// TwinCAT 3 PLC project FastLog
// ProgramVersion: 3.1.4024.0
// libraries:
//   Tc2_Standard, * (Beckhoff Automation GmbH)
//   Tc2_System, * (Beckhoff Automation GmbH)
//   Tc2_Utilities, * (Beckhoff Automation GmbH)
//   Tc3_Module, * (Beckhoff Automation GmbH)
// project tree:
//   / FileLogger.TcTTO, FastSample.TcTTO
//   GVLs/ GVL.TcGVL, SENSOR_LIST.TcGVL
//   POUs/ F_TimeStructToUnixMs.TcPOU, PRG_FileLogger.TcPOU, PRG_FastSample.TcPOU
// real-time tasks:
//   TASK FastSample: cycle T#100us, priority 20, ADS port 350
//   TASK FileLogger: cycle T#1ms, priority 10, ADS port 351
// I/O:
//   DEVICE Device 1 (Beckhoff CCAT)
//   DEVICE Device 2 (EtherCAT), AmsNetId 5.156.10.9.3.1
//     Term 1 (EK1200) [EK1200-5000 EtherCAT Power supply (2A E-Bus)]
//       Term 2 (EL1809) [EL1809 16Ch. Dig. Input 24V, 3ms]
//       Term 3 (EL1889) [EL1889 16Ch. Dig. Input 24V, 3ms, negative]
//       Term 4 (EL2008) [EL2008 8Ch. Dig. Output 24V, 0.5A]
//       Term 5 (EL2008) [EL2008 8Ch. Dig. Output 24V, 0.5A]
//       Term 6 (EL2008) [EL2008 8Ch. Dig. Output 24V, 0.5A]
//       Term 7 (EL2634) [EL2634 4Ch. Relay Output, NO (250V AC / 30V DC)]
//       Term 8 (EL2889) [EL2889 16Ch. Dig. Output 24V, 0.5A, negative]
//       Term 9 (EL2809) [EL2809 16Ch. Dig. Output 24V, 0.5A]
//       Term 10 (EL9011) [EL9011 End Terminal]
//   DEVICE Device 5 (EtherCAT), AmsNetId 5.156.10.9.6.1
//     Term 11 (EK1100) [EK1100 EtherCAT Coupler (2A E-Bus)]
//       Term 12 (EL5151) [EL5151 1Ch. Inc. Encoder]
//       Term 13 (EL5151) [EL5151 1Ch. Inc. Encoder]
//       Term 14 (EL3182) [EL3182 2Ch. Ana. Input 4-20mA, HART]
//         modules: Ch. 1, Ch. 2, Ch. 1, Ch. 1, Ch. 1, Ch. 1, Ch. 1, Ch. 1, Ch. 1, Ch. 1, Ch. 1, Ch. 1, Ch. 1, Ch. 1, Ch. 1
//       Term 15 (EL3182) [EL3182 2Ch. Ana. Input 4-20mA, HART]
//         modules: Ch. 1, Ch. 2, Ch. 1, Ch. 1, Ch. 1, Ch. 1, Ch. 1, Ch. 1, Ch. 1, Ch. 1, Ch. 1, Ch. 1, Ch. 1, Ch. 1, Ch. 1
//       Term 6 (EL6731) [EL6731 PROFIBUS DP Master]
//       Term 7 (EL6751) [EL6751 CANopen Master]
//       Term 18 (EL6022) [EL6022 Interface 2Ch. (RS422/485)]
//       Term 19 (EL6022) [EL6022 Interface 2Ch. (RS422/485)]
//       Term 62 (EL9011) [EL9011 End Terminal]
//     Term 20 (EK1100) [EK1100 EtherCAT Coupler (2A E-Bus)]
//       Term 21 (EL3201-0020) [EL3201-0020 1Ch. Ana. Input PT100 (RTD), High Precision, calibrated]
//       Term 22 (EL3201-0020) [EL3201-0020 1Ch. Ana. Input PT100 (RTD), High Precision, calibrated]
//       Term 23 (EL3201-0020) [EL3201-0020 1Ch. Ana. Input PT100 (RTD), High Precision, calibrated]
//       Term 24 (EL3201-0020) [EL3201-0020 1Ch. Ana. Input PT100 (RTD), High Precision, calibrated]
//       Term 25 (EL3201-0020) [EL3201-0020 1Ch. Ana. Input PT100 (RTD), High Precision, calibrated]
//       Term 26 (EL3201-0020) [EL3201-0020 1Ch. Ana. Input PT100 (RTD), High Precision, calibrated]
//       Term 27 (EL3201-0020) [EL3201-0020 1Ch. Ana. Input PT100 (RTD), High Precision, calibrated]
//       Term 28 (EL3201-0020) [EL3201-0020 1Ch. Ana. Input PT100 (RTD), High Precision, calibrated]
//       Term 29 (EL3201-0020) [EL3201-0020 1Ch. Ana. Input PT100 (RTD), High Precision, calibrated]
//       Term 30 (EL9410) [EL9410 E-Bus Power Supplier  (Diagnostics)]
//       Term 31 (EL3201-0020) [EL3201-0020 1Ch. Ana. Input PT100 (RTD), High Precision, calibrated]
//       Term 32 (EL3201-0020) [EL3201-0020 1Ch. Ana. Input PT100 (RTD), High Precision, calibrated]
//       Term 33 (EL3201-0020) [EL3201-0020 1Ch. Ana. Input PT100 (RTD), High Precision, calibrated]
//       Term 34 (EL3201-0020) [EL3201-0020 1Ch. Ana. Input PT100 (RTD), High Precision, calibrated]
//       Term 35 (EL3201-0020) [EL3201-0020 1Ch. Ana. Input PT100 (RTD), High Precision, calibrated]
//       Term 36 (EL3201-0020) [EL3201-0020 1Ch. Ana. Input PT100 (RTD), High Precision, calibrated]
//       Term 37 (EL3201-0020) [EL3201-0020 1Ch. Ana. Input PT100 (RTD), High Precision, calibrated]
//       Term 38 (EL3218) [EL3218-0000 8Ch. Ana. Input PT100 (RTD)]
//       Term 39 (EL3218) [EL3218-0000 8Ch. Ana. Input PT100 (RTD)]
//       Term 40 (EL3218) [EL3218-0000 8Ch. Ana. Input PT100 (RTD)]
//       Term 41 (EL9410) [EL9410 E-Bus Power Supplier  (Diagnostics)]
//       Term 42 (EL3218) [EL3218-0000 8Ch. Ana. Input PT100 (RTD)]
//       Term 43 (EL3218) [EL3218-0000 8Ch. Ana. Input PT100 (RTD)]
//       Term 44 (EL3218) [EL3218-0000 8Ch. Ana. Input PT100 (RTD)]
//       Term 45 (EL3214) [EL3214 4Ch. Ana. Input PT100 (RTD)]
//       Term 46 (EL4124) [EL4124 4Ch. Ana. Output 4-20mA, 16bit]
//       Term 47 (EL4124) [EL4124 4Ch. Ana. Output 4-20mA, 16bit]
//       Term 48 (EL4124) [EL4124 4Ch. Ana. Output 4-20mA, 16bit]
//       Term 49 (EL4124) [EL4124 4Ch. Ana. Output 4-20mA, 16bit]
//       Term 50 (EL4124) [EL4124 4Ch. Ana. Output 4-20mA, 16bit]
//       Term 51 (EL4124) [EL4124 4Ch. Ana. Output 4-20mA, 16bit]
//       Term 52 (EL4124) [EL4124 4Ch. Ana. Output 4-20mA, 16bit]
//       Term 53 (EL3356) [EL3356 1Ch. Ana. Input Resistor Bridge Terminal, 16bit, High Precision]
//       Term 63 (EL9011) [EL9011 End Terminal]
//     Term 54 (EK1100) [EK1100 EtherCAT Coupler (2A E-Bus)]
//       Term 55 (ELM3148-0000) [ELM3148-0000 8Ch. Ana. Input +/-10V, +/-20mA, 24 bit, high precision]
//       Term 56 (ELM3148-0000) [ELM3148-0000 8Ch. Ana. Input +/-10V, +/-20mA, 24 bit, high precision]
//       Term 57 (ELM3148-0000) [ELM3148-0000 8Ch. Ana. Input +/-10V, +/-20mA, 24 bit, high precision]
//       Term 58 (ELM3148-0000) [ELM3148-0000 8Ch. Ana. Input +/-10V, +/-20mA, 24 bit, high precision]
//       Term 59 (ELM3148-0000) [ELM3148-0000 8Ch. Ana. Input +/-10V, +/-20mA, 24 bit, high precision]
//       Term 60 (ELM3148-0000) [ELM3148-0000 8Ch. Ana. Input +/-10V, +/-20mA, 24 bit, high precision]
//       Term 61 (EL9410) [EL9410 E-Bus Power Supplier  (Diagnostics)]
//       Term 62 (ELM3148-0000) [ELM3148-0000 8Ch. Ana. Input +/-10V, +/-20mA, 24 bit, high precision]
//       Term 63 (ELM3148-0000) [ELM3148-0000 8Ch. Ana. Input +/-10V, +/-20mA, 24 bit, high precision]
//       Term 64 (ELM3148-0000) [ELM3148-0000 8Ch. Ana. Input +/-10V, +/-20mA, 24 bit, high precision]
//       Term 65 (ELM3148-0000) [ELM3148-0000 8Ch. Ana. Input +/-10V, +/-20mA, 24 bit, high precision]
//       Term 66 (ELM3148-0000) [ELM3148-0000 8Ch. Ana. Input +/-10V, +/-20mA, 24 bit, high precision]
//       Term 67 (ELM3148-0000) [ELM3148-0000 8Ch. Ana. Input +/-10V, +/-20mA, 24 bit, high precision]
//       Term 68 (EL9410) [EL9410 E-Bus Power Supplier  (Diagnostics)]
//       Term 69 (ELM3148-0000) [ELM3148-0000 8Ch. Ana. Input +/-10V, +/-20mA, 24 bit, high precision]
//       Term 70 (ELM3148-0000) [ELM3148-0000 8Ch. Ana. Input +/-10V, +/-20mA, 24 bit, high precision]
//       Term 71 (ELM3148-0000) [ELM3148-0000 8Ch. Ana. Input +/-10V, +/-20mA, 24 bit, high precision]
//       Term 64 (EL9011) [EL9011 End Terminal]
//   DEVICE Device 6 (USB)
//     Box 1 (CX2100 Power Supply)
//   DEVICE Device 7 (NOV-DP-RAM)
//   DEVICE Device 3 (EL6731), AmsNetId 5.156.10.9.4.1
//   DEVICE Device 4 (EL6751), AmsNetId 5.156.10.9.5.1
// variable links:
//   FastLog/FastLog Instance <-> Device 5 (EtherCAT)/Term 54 (EK1100)/Term 55 (ELM3148-0000)
//     FastSample Inputs/SENSOR_LIST.AInput_{1..8} <-> PAI Samples 1 Channel {1..8}/Samples[0]  (8 links)
//   FastLog/FastLog Instance <-> Device 5 (EtherCAT)/Term 54 (EK1100)/Term 56 (ELM3148-0000)
//     FastSample Inputs/SENSOR_LIST.AInput_{9..16} <-> PAI Samples 1 Channel {1..8}/Samples[0]  (8 links)
//   FastLog/FastLog Instance <-> Device 5 (EtherCAT)/Term 54 (EK1100)/Term 57 (ELM3148-0000)
//     FastSample Inputs/SENSOR_LIST.AInput_17 <-> PAI Samples 1 Channel 1/Samples[0]
//     FastSample Inputs/SENSOR_LIST.AInput_18 <-> PAI Samples 1 Channel 2/Samples[0]
//     FastSample Inputs/SENSOR_LIST.AInput_19 <-> PAI Samples 1 Channel 3/Samples[0]
//     FastSample Inputs/SENSOR_LIST.AInput_20 <-> PAI Samples 1 Channel 4/Samples[0]
//     FastSample Inputs/SENSOR_LIST.AInput_21 <-> PAI Samples 1 Channel 5/Samples[0]
//     FastSample Inputs/SENSOR_LIST.AInput_22 <-> PAI Samples 1 Channel 6/Samples[0]
//     FastSample Inputs/SENSOR_LIST.AInput_24 <-> PAI Samples 1 Channel 8/Samples[0]
//     FastSample Inputs/SENSOR_LIST.AInput_23 <-> PAI Samples 1 Channel 7/Samples

CONFIGURATION FastLog
    RESOURCE PLC ON TwinCAT3
        TASK FileLogger(INTERVAL := T#100us, PRIORITY := 20);
        TASK FastSample(INTERVAL := T#1ms, PRIORITY := 10);
        PROGRAM PRG_FileLogger WITH FileLogger : PRG_FileLogger;
        PROGRAM PRG_FastSample WITH FastSample : PRG_FastSample;
    END_RESOURCE
END_CONFIGURATION

// ---- GVLs/GVL.TcGVL
VAR_GLOBAL CONSTANT
    C_BUFFER_SIZE : UDINT := 100000;   // buffer satır sayısı (ihtiyacına göre büyüt)
    C_NUM_SENSORS : UINT  := 60;       // sende 60 sensör var demiştin
END_VAR


VAR_GLOBAL
    // Start/Stop
    g_bLogStart       : BOOL := FALSE;
    g_bLogStop        : BOOL := FALSE;
    g_bLogging        : BOOL := FALSE;

    // Epoch ms (sampler doldurur)
    g_epochMs        : ULINT := 0;
	g_epochBaseMs    : ULINT := 0;   // log start anındaki gerçek epoch(ms)
    g_epochOffsetMs  : UDINT := 0; 

    // Ring buffer
    g_aTimeBuffer     : ARRAY[0..C_BUFFER_SIZE-1] OF ULINT;
    g_aValBuffer      : ARRAY[0..C_BUFFER_SIZE-1, 1..C_NUM_SENSORS] OF LREAL;

    g_wrIndex         : UDINT := 0;
    g_rdIndex         : UDINT := 0;
    g_bufferUsed      : UDINT := 0;
    g_bufferOverflow  : BOOL  := FALSE;

    // Sampler burayı dolduracak
    g_arCurrentValues : ARRAY[1..C_NUM_SENSORS] OF LREAL;

    // Dosya yolu / isim
    g_sBasePath       : STRING(255) := 'D:\';   // istediğin klasör
    g_sFileName       : STRING(64);
    g_sPath           : STRING(320);

    // Yazma kontrol
    g_headerPending   : BOOL := FALSE;
    g_lineReady       : BOOL := FALSE;

    // Chunk buffer (data satırları buraya toplanır)
    g_sLine           : STRING(16384);

END_VAR

// ---- GVLs/SENSOR_LIST.TcGVL
VAR_GLOBAL
	
	AInput_1  AT %I* : DINT;
	AInput_2  AT %I* : DINT;
	AInput_3  AT %I* : DINT;
	AInput_4  AT %I* : DINT;
	AInput_5  AT %I* : DINT;
	AInput_6  AT %I* : DINT;
	AInput_7  AT %I* : DINT;
	AInput_8  AT %I* : DINT;
	AInput_9  AT %I* : DINT;
	AInput_10 AT %I* : DINT;
	AInput_11 AT %I* : DINT;
	AInput_12 AT %I* : DINT;
	AInput_13 AT %I* : DINT;
	AInput_14 AT %I* : DINT;
	AInput_15 AT %I* : DINT;
	AInput_16 AT %I* : DINT;
	AInput_17 AT %I* : DINT;
	AInput_18 AT %I* : DINT;
	AInput_19 AT %I* : DINT;
	AInput_20 AT %I* : DINT;
	
	AInput_21 AT %I* : DINT;
	AInput_22 AT %I* : DINT;
	AInput_23 AT %I* : DINT;
	AInput_24 AT %I* : DINT;
	AInput_25 AT %I* : DINT;
	AInput_26 AT %I* : DINT;
	AInput_27 AT %I* : DINT;
	AInput_28 AT %I* : DINT;
	AInput_29 AT %I* : DINT;
	AInput_30 AT %I* : DINT;
	
	AInput_31 AT %I* : DINT;
	AInput_32 AT %I* : DINT;
	AInput_33 AT %I* : DINT;
	AInput_34 AT %I* : DINT;
	AInput_35 AT %I* : DINT;
	AInput_36 AT %I* : DINT;
	AInput_37 AT %I* : DINT;
	AInput_38 AT %I* : DINT;
	AInput_39 AT %I* : DINT;
	AInput_40 AT %I* : DINT;
	
	AInput_41 AT %I* : DINT;
	AInput_42 AT %I* : DINT;
	AInput_43 AT %I* : DINT;
	AInput_44 AT %I* : DINT;
	AInput_45 AT %I* : DINT;
	AInput_46 AT %I* : DINT;
	AInput_47 AT %I* : DINT;
	AInput_48 AT %I* : DINT;
	AInput_49 AT %I* : DINT;
	AInput_50 AT %I* : DINT;
	
	AInput_51 AT %I* : DINT;
	AInput_52 AT %I* : DINT;
	AInput_53 AT %I* : DINT;
	AInput_54 AT %I* : DINT;
	AInput_55 AT %I* : DINT;
	AInput_56 AT %I* : DINT;
	AInput_57 AT %I* : DINT;
	AInput_58 AT %I* : DINT;
	AInput_59 AT %I* : DINT;
	AInput_60 AT %I* : DINT;

END_VAR

// ---- POUs/PRG_FileLogger.TcPOU
PROGRAM PRG_FileLogger
VAR
    // Start/Stop edge
    bLogStartOld   : BOOL := FALSE;
    bLogStopOld    : BOOL := FALSE;

    // Saat
    fbLocalTime    : Tc2_Utilities.FB_LocalSystemTime;
    tsNow          : TIMESTRUCT;

    // File FB'leri
    fbOpen         : FB_FileOpen;
    fbWrite        : FB_FileWrite;
    fbClose        : FB_FileClose;
    hFile          : UINT := 0;

    // State machine
    fileState      : INT := 0;   // 0 idle, 10 open, 30 log, 90 close
    writeState     : INT := 0;   // 0 idle, 1 start write, 2 wait

    // Chunk ayarları
    C_CHUNK_SIZE   : UINT := 50;
    chunkCount     : UINT := 0;
    idx            : UDINT;
    iSens          : UINT;

    // küçük string parçaları (255 altı!)
    sPiece         : STRING(80);

    // BYTE buffer (uzun satırlar burada)
    aBuf           : ARRAY[0..16383] OF BYTE;   // 16 KB
    nBufLen        : UDINT := 0;

    // Yazılacak buffer seçimi
    pWriteBuff     : PVOID;
    nWriteLen      : UDINT;
END_VAR

// =============================
// PLC saatini sürekli güncelle
// =============================
fbLocalTime(bEnable := TRUE);
fbLocalTime();
IF fbLocalTime.bValid THEN
    tsNow := fbLocalTime.systemTime;
END_IF;


// =============================
// Start / Stop edge detect
// =============================
IF g_bLogStart AND NOT bLogStartOld THEN
    g_bLogging       := TRUE;
    g_epochOffsetMs  := 0;
    g_wrIndex        := 0;
    g_rdIndex        := 0;
    g_bufferOverflow := FALSE;
    
    // Log başlangıcında base epoch (eğer kullanıyorsan)
    g_epochBaseMs := F_TimeStructToUnixMs(tsNow);

    // Dosya ismi
    g_sFileName := UINT_TO_STRING(tsNow.wDay);
    g_sFileName := CONCAT(g_sFileName, UINT_TO_STRING(tsNow.wMonth));
    g_sFileName := CONCAT(g_sFileName, UINT_TO_STRING(tsNow.wYear MOD 100));
    g_sFileName := CONCAT(g_sFileName, '-');
    g_sFileName := CONCAT(g_sFileName, UINT_TO_STRING(tsNow.wHour));
    g_sFileName := CONCAT(g_sFileName, '_');
    g_sFileName := CONCAT(g_sFileName, UINT_TO_STRING(tsNow.wMinute));
    g_sFileName := CONCAT(g_sFileName, '_');
    g_sFileName := CONCAT(g_sFileName, UINT_TO_STRING(tsNow.wSecond));
    g_sFileName := CONCAT(g_sFileName, '.csv');

    g_sPath := CONCAT(g_sBasePath, g_sFileName);

    g_headerPending := TRUE;
    g_lineReady     := FALSE;

    writeState := 0;
    fileState  := 10;
END_IF;

IF g_bLogStop AND NOT bLogStopOld THEN
    g_bLogging := FALSE;
END_IF;

bLogStartOld := g_bLogStart;
bLogStopOld  := g_bLogStop;


// =============================
// DOSYA / YAZMA STATE MACHINE
// =============================
CASE fileState OF

    0: ; // IDLE

    // -------------------------
    // 10: Dosyayı aç
    // -------------------------
    10:
        fbOpen.sNetId    := '';
        fbOpen.sPathName := g_sPath;
        fbOpen.nMode     := FOPEN_MODEWRITE OR FOPEN_MODETEXT; // CREATE yok, WRITE yeterli
        fbOpen.bExecute  := TRUE;
        fbOpen();
        fbOpen.bExecute  := FALSE;
        fileState := 11;

    11:
        fbOpen();
        IF NOT fbOpen.bBusy THEN
            IF fbOpen.bError THEN
                fileState := 0;
            ELSE
                hFile := fbOpen.hFile;
                fileState := 30;
            END_IF
        END_IF


    // -------------------------
    // 30: LOGGING
    // -------------------------
    30:
        // ---- A) Yazma state ----
        CASE writeState OF
            0:
                IF g_lineReady THEN
                    writeState := 1;
                END_IF

            1:
                fbWrite.sNetId     := '';
                fbWrite.hFile      := hFile;
                fbWrite.pWriteBuff := pWriteBuff;
                fbWrite.cbWriteLen := nWriteLen;
                fbWrite.bExecute   := TRUE;
                fbWrite();
                fbWrite.bExecute   := FALSE;
                writeState := 2;

            2:
                fbWrite();
                IF NOT fbWrite.bBusy THEN
                    g_lineReady := FALSE;
                    writeState  := 0;
                END_IF
        END_CASE


        // ---- B) Yeni yazılacak şey hazırla ----
        IF (writeState = 0) AND (NOT g_lineReady) THEN

            // ======================
            // 1) HEADER (BYTE buffer)
            // ======================
            IF g_headerPending THEN

                nBufLen := 0;

                // "TimeMs" (aslında EpochMs yazmak istersen burayı değiştir)
                sPiece := 'TimeMs';
                MEMCPY(ADR(aBuf[nBufLen]), ADR(sPiece), LEN(sPiece));
                nBufLen := nBufLen + LEN(sPiece);

                // ",ValueX" kolonları
                FOR iSens := 1 TO C_NUM_SENSORS DO
                    sPiece := ',Value';
                    sPiece := CONCAT(sPiece, UINT_TO_STRING(iSens));
                    MEMCPY(ADR(aBuf[nBufLen]), ADR(sPiece), LEN(sPiece));
                    nBufLen := nBufLen + LEN(sPiece);
                END_FOR

                // newline
                sPiece := '$N';
                MEMCPY(ADR(aBuf[nBufLen]), ADR(sPiece), LEN(sPiece));
                nBufLen := nBufLen + LEN(sPiece);

                pWriteBuff  := ADR(aBuf);
                nWriteLen   := nBufLen;
                g_lineReady := TRUE;

                g_headerPending := FALSE;

            ELSE

                // ======================
                // 2) DATA CHUNK (BYTE buffer)
                // ======================
                g_bufferUsed := g_wrIndex - g_rdIndex;

                IF g_bufferUsed > 0 THEN
                    nBufLen    := 0;
                    chunkCount := 0;

                    WHILE (chunkCount < C_CHUNK_SIZE) AND (g_rdIndex < g_wrIndex) DO
                        // 🔴 ÖNEMLİ: index artık UDINT, cast yok
                        idx := g_rdIndex MOD C_BUFFER_SIZE;

                        // TimeMs / EpochMs
                        sPiece := ULINT_TO_STRING(g_aTimeBuffer[idx]);
                        MEMCPY(ADR(aBuf[nBufLen]), ADR(sPiece), LEN(sPiece));
                        nBufLen := nBufLen + LEN(sPiece);

                        // tüm sensörler
                        FOR iSens := 1 TO C_NUM_SENSORS DO
                            sPiece := ',';
                            MEMCPY(ADR(aBuf[nBufLen]), ADR(sPiece), LEN(sPiece));
                            nBufLen := nBufLen + LEN(sPiece);

                            sPiece := LREAL_TO_STRING(g_aValBuffer[idx, iSens]);
                            MEMCPY(ADR(aBuf[nBufLen]), ADR(sPiece), LEN(sPiece));
                            nBufLen := nBufLen + LEN(sPiece);
                        END_FOR

                        // newline
                        sPiece := '$N';
                        MEMCPY(ADR(aBuf[nBufLen]), ADR(sPiece), LEN(sPiece));
                        nBufLen := nBufLen + LEN(sPiece);

                        g_rdIndex  := g_rdIndex + 1;
                        chunkCount := chunkCount + 1;

                        // buffer taşmasın – aBuf en az 16000 ise 15000 sınırı güvenli
                        IF nBufLen > 15000 THEN
                            EXIT;
                        END_IF
                    END_WHILE

                    pWriteBuff  := ADR(aBuf);
                    nWriteLen   := nBufLen;
                    g_lineReady := TRUE;

                ELSE
                    // Buffer boş & logging de OFF ise → dosyayı kapat
                    IF NOT g_bLogging THEN
                        fileState := 90;
                    END_IF
                END_IF
            END_IF
        END_IF


    // -------------------------
    // 90: Dosyayı kapat
    // -------------------------
    90:
        fbClose.sNetId   := '';
        fbClose.hFile    := hFile;
        fbClose.bExecute := TRUE;
        fbClose();
        fbClose.bExecute := FALSE;
        fileState := 91;

    91:
        fbClose();
        IF NOT fbClose.bBusy THEN
            hFile    := 0;
            fileState := 0;
        END_IF

END_CASE

END_PROGRAM

// ---- POUs/F_TimeStructToUnixMs.TcPOU
FUNCTION F_TimeStructToUnixMs : ULINT
VAR_INPUT
    ts : TIMESTRUCT;
END_VAR
VAR
    y         : UDINT;
    m         : UDINT;
    d         : UDINT;
    days      : ULINT;
    i         : UDINT;
    leap      : BOOL;
    mdays     : ARRAY[1..12] OF UDINT := [31,28,31,30,31,30,31,31,30,31,30,31];
END_VAR

// yılı 2000+ kabul ediyoruz (TIMESTRUCT wYear zaten 4 haneli)
y := TO_UDINT(ts.wYear);
m := TO_UDINT(ts.wMonth);
d := TO_UDINT(ts.wDay);

// Leap year kontrolü
leap := ( (y MOD 4 = 0) AND (y MOD 100 <> 0) ) OR (y MOD 400 = 0);

// 1970'ten önceyse 0 dön (fazla uğraşmayalım)
IF y < 1970 THEN
    F_TimeStructToUnixMs := 0;
    RETURN;
END_IF;

// year days
days := 0;
FOR i := 1970 TO y-1 DO
    IF ( (i MOD 4 = 0) AND (i MOD 100 <> 0) ) OR (i MOD 400 = 0) THEN
        days := days + 366;
    ELSE
        days := days + 365;
    END_IF
END_FOR

// month days
FOR i := 1 TO m-1 DO
    days := days + mdays[i];
    IF (i = 2) AND leap THEN
        days := days + 1;
    END_IF
END_FOR

// day index
days := days + (d - 1);

// ms
F_TimeStructToUnixMs :=
    days * 86400000
  + TO_ULINT(ts.wHour)       * 3600000
  + TO_ULINT(ts.wMinute)     * 60000
  + TO_ULINT(ts.wSecond)     * 1000
  + TO_ULINT(ts.wMilliseconds);

END_FUNCTION

// ---- POUs/PRG_FastSample.TcPOU
PROGRAM PRG_FastSample
VAR
    idxBuf : UDINT;
    iSens  : UINT;
	fbLT   : Tc2_Utilities.FB_LocalSystemTime;
    ts     : TIMESTRUCT;
    lastMs : UDINT := 0;
    nowMs  : UDINT := 0;
    dMs    : UDINT := 0;
    g_dbgAvgMs : LREAL := 0;  // GVL'e koyarsan izlersin
	epochNow : ULINT;
    epochMs : ULINT;

END_VAR

// =============================
// Sistem zamanını oku (tek sefer)
// =============================
fbLT(bEnable := TRUE);
fbLT();

IF fbLT.bValid THEN
    ts := fbLT.systemTime;

    // ---- 1) EPOCH (ms since 1970) hesapla ----
    epochMs := F_TimeStructToUnixMs(ts);

    // ---- 2) Debug için gerçek ms farkını hesapla (opsiyonel) ----
    nowMs := TO_UDINT(ts.wHour) * 3600000
           + TO_UDINT(ts.wMinute) * 60000
           + TO_UDINT(ts.wSecond) * 1000
           + TO_UDINT(ts.wMilliseconds);

    IF lastMs <> 0 THEN
        dMs := nowMs - lastMs;
        // son 100 örneğin ortalaması (LREAL)
        g_dbgAvgMs := (g_dbgAvgMs * 99.0 + TO_LREAL(dMs)) / 100.0;
    END_IF;

    lastMs := nowMs;
END_IF;


// =============================
// Örnek alma (logging açıkken)
// =============================
IF g_bLogging AND fbLT.bValid THEN

    // 1) Ring buffer index
    idxBuf := g_wrIndex MOD C_BUFFER_SIZE;

    // 2) Zamanı yaz (epoch ms -> ULINT)
    g_aTimeBuffer[idxBuf] := epochMs;

    // 3) Sensörleri oku -> g_arCurrentValues[...] doldur
    g_arCurrentValues[1]  := DINT_TO_LREAL(SENSOR_LIST.AInput_1);
    g_arCurrentValues[2]  := DINT_TO_LREAL(SENSOR_LIST.AInput_2);
    g_arCurrentValues[3]  := DINT_TO_LREAL(SENSOR_LIST.AInput_3);
    g_arCurrentValues[4]  := DINT_TO_LREAL(SENSOR_LIST.AInput_4);
    g_arCurrentValues[5]  := DINT_TO_LREAL(SENSOR_LIST.AInput_5);
    g_arCurrentValues[6]  := DINT_TO_LREAL(SENSOR_LIST.AInput_6);
    g_arCurrentValues[7]  := DINT_TO_LREAL(SENSOR_LIST.AInput_7);
    g_arCurrentValues[8]  := DINT_TO_LREAL(SENSOR_LIST.AInput_8);
    g_arCurrentValues[9]  := DINT_TO_LREAL(SENSOR_LIST.AInput_9);
    g_arCurrentValues[10] := DINT_TO_LREAL(SENSOR_LIST.AInput_10);
    
    g_arCurrentValues[11] := DINT_TO_LREAL(SENSOR_LIST.AInput_11);
    g_arCurrentValues[12] := DINT_TO_LREAL(SENSOR_LIST.AInput_12);
    g_arCurrentValues[13] := DINT_TO_LREAL(SENSOR_LIST.AInput_13);
    g_arCurrentValues[14] := DINT_TO_LREAL(SENSOR_LIST.AInput_14);
    g_arCurrentValues[15] := DINT_TO_LREAL(SENSOR_LIST.AInput_15);
    g_arCurrentValues[16] := DINT_TO_LREAL(SENSOR_LIST.AInput_16);
    g_arCurrentValues[17] := DINT_TO_LREAL(SENSOR_LIST.AInput_17);
    g_arCurrentValues[18] := DINT_TO_LREAL(SENSOR_LIST.AInput_18);
    g_arCurrentValues[19] := DINT_TO_LREAL(SENSOR_LIST.AInput_19);
    g_arCurrentValues[20] := DINT_TO_LREAL(SENSOR_LIST.AInput_20);
    
    g_arCurrentValues[21] := DINT_TO_LREAL(SENSOR_LIST.AInput_21);
    g_arCurrentValues[22] := DINT_TO_LREAL(SENSOR_LIST.AInput_22);
    g_arCurrentValues[23] := DINT_TO_LREAL(SENSOR_LIST.AInput_23);
    g_arCurrentValues[24] := DINT_TO_LREAL(SENSOR_LIST.AInput_24);
    g_arCurrentValues[25] := DINT_TO_LREAL(SENSOR_LIST.AInput_25);
    g_arCurrentValues[26] := DINT_TO_LREAL(SENSOR_LIST.AInput_26);
    g_arCurrentValues[27] := DINT_TO_LREAL(SENSOR_LIST.AInput_27);
    g_arCurrentValues[28] := DINT_TO_LREAL(SENSOR_LIST.AInput_28);
    g_arCurrentValues[29] := DINT_TO_LREAL(SENSOR_LIST.AInput_29);
    g_arCurrentValues[30] := DINT_TO_LREAL(SENSOR_LIST.AInput_30);
    
    g_arCurrentValues[31] := DINT_TO_LREAL(SENSOR_LIST.AInput_31);
    g_arCurrentValues[32] := DINT_TO_LREAL(SENSOR_LIST.AInput_32);
    g_arCurrentValues[33] := DINT_TO_LREAL(SENSOR_LIST.AInput_33);
    g_arCurrentValues[34] := DINT_TO_LREAL(SENSOR_LIST.AInput_34);
    g_arCurrentValues[35] := DINT_TO_LREAL(SENSOR_LIST.AInput_35);
    g_arCurrentValues[36] := DINT_TO_LREAL(SENSOR_LIST.AInput_36);
    g_arCurrentValues[37] := DINT_TO_LREAL(SENSOR_LIST.AInput_37);
    g_arCurrentValues[38] := DINT_TO_LREAL(SENSOR_LIST.AInput_38);
    g_arCurrentValues[39] := DINT_TO_LREAL(SENSOR_LIST.AInput_39);
    g_arCurrentValues[40] := DINT_TO_LREAL(SENSOR_LIST.AInput_40);
    
    g_arCurrentValues[41] := DINT_TO_LREAL(SENSOR_LIST.AInput_41);
    g_arCurrentValues[42] := DINT_TO_LREAL(SENSOR_LIST.AInput_42);
    g_arCurrentValues[43] := DINT_TO_LREAL(SENSOR_LIST.AInput_43);
    g_arCurrentValues[44] := DINT_TO_LREAL(SENSOR_LIST.AInput_44);
    g_arCurrentValues[45] := DINT_TO_LREAL(SENSOR_LIST.AInput_45);
    g_arCurrentValues[46] := DINT_TO_LREAL(SENSOR_LIST.AInput_46);
    g_arCurrentValues[47] := DINT_TO_LREAL(SENSOR_LIST.AInput_47);
    g_arCurrentValues[48] := DINT_TO_LREAL(SENSOR_LIST.AInput_48);
    g_arCurrentValues[49] := DINT_TO_LREAL(SENSOR_LIST.AInput_49);
    g_arCurrentValues[50] := DINT_TO_LREAL(SENSOR_LIST.AInput_50);
    
    g_arCurrentValues[51] := DINT_TO_LREAL(SENSOR_LIST.AInput_51);
    g_arCurrentValues[52] := DINT_TO_LREAL(SENSOR_LIST.AInput_52);
    g_arCurrentValues[53] := DINT_TO_LREAL(SENSOR_LIST.AInput_53);
    g_arCurrentValues[54] := DINT_TO_LREAL(SENSOR_LIST.AInput_54);
    g_arCurrentValues[55] := DINT_TO_LREAL(SENSOR_LIST.AInput_55);
    g_arCurrentValues[56] := DINT_TO_LREAL(SENSOR_LIST.AInput_56);
    g_arCurrentValues[57] := DINT_TO_LREAL(SENSOR_LIST.AInput_57);
    g_arCurrentValues[58] := DINT_TO_LREAL(SENSOR_LIST.AInput_58);
    g_arCurrentValues[59] := DINT_TO_LREAL(SENSOR_LIST.AInput_59);
    g_arCurrentValues[60] := DINT_TO_LREAL(SENSOR_LIST.AInput_60);

    // 4) Buffer doluluk kontrolü ve yazma
    g_bufferUsed := g_wrIndex - g_rdIndex;

    IF g_bufferUsed < C_BUFFER_SIZE THEN
        // sensörleri buffer'a kopyala
        FOR iSens := 1 TO C_NUM_SENSORS DO
            g_aValBuffer[idxBuf, iSens] := g_arCurrentValues[iSens];
        END_FOR;

        g_wrIndex := g_wrIndex + 1;
    ELSE
        g_bufferOverflow := TRUE;   // logger yetişemiyor
        g_bLogging := FALSE;        // istersen burada sampling'i de durdur
    END_IF;

END_IF;

END_PROGRAM
